# EPICS autosave request: iocMythen/auto_settings.req
$(P)cam1:AcquireTime.PREC
file "mythen_settings.req",       P=$(P),  R=cam1:
file "NDStdArrays_settings.req",  P=$(P),  R=image1:
file "commonPlugin_settings.req", P=$(P)
